          case 6
            call UI:Control_YesNO("确定需要关门吗？",l_bRes)
            if l_bRes
              call UI:Control_PanelMd("正在关闭门....")
              if x_b8Axis
                call IO:AxisDoor(false,true)
              else
                call IO:AxisDoor(false,false)
              endIf
            endIf
            cls()
          break

          //刷新当前轴值
          case 7


          break


        endSwitch


      break

      case -1

        if x_b8Axis
          call IO:Axis8Action(9)
        else
          call IO:Axis7Action(9)
        endIf

      break

    endSwitch



    //当前七轴位置
    if l_nKey!=-1 or !l_bFirst


      //


      l_bFirst=true
      gotoxy(0,0)
      put("运动机械手臂须上电     ")

      //××××××××××××××××××××××××××××


      sSItem[0]="位置mm   :"+toString(".3",l_nPosition)
      sSItem[1]="速度m/min:"+toString(".3",l_nSpeed)
      sSItem[2]="比例分度 :"+toString("",l_nPrecent)
      sSItem[3]="点动速度 :"+toString("",l_nJogSpeed)+"%"
      sSItem[4]="报警复位"
      sSItem[5]="门打开"
      sSItem[6]="门关闭"
      //sSItem[7]="当前马达值"
      if bCheckAxisSafte
        l_sBottom="+,-,,回零,运动,,,退出"
      else
        l_sBottom="+,-,记录,回零,运动,上传,保存,退出"
      endIf
      if !x_b8Axis

        call UI:Form_PanelList("LasMAN3.6->示教异步七轴","第七轴",sSItem,l_nIndex,l_sBottom)

      else
        call UI:Form_PanelList("LasMAN3.6->示教异步八轴","第八轴",sSItem,l_nIndex,l_sBottom)

      endIf


    endIf


    //报警处理
    if l_bAlarm
      call UI:Control_Mess("马达报警            ","")
    else
      if !l_bPowerOn
        if l_bBHome
          call UI:Control_Mess("马达已回零,未上电","")
        else
          call UI:Control_Mess("马达未回零,未上电","")
        endIf
      else
        if l_bBHome
          setTextMode(0)
          call UI:Control_Mess("马达已回零,已上电","")
        else
          call UI:Control_Mess("马达未回零,已上电","")
        endIf
      endIf

    endIf




    //2014.08.04
    //实时显示异步七轴八轴位置

    if l_bAlarm==false and l_bPowerOn==true
      if x_b8Axis
        call IO:GetAxis8Pos(l_nBuff,l_nPrecent)
      else
        call IO:GetAxis7Pos(l_nBuff,l_nPrecent)
      endIf
      gotoxy(0,2)
      put("轴当前位置:"+toString(".3",l_nBuff)+"     ")
    endIf
    delay(0)

  endWhile


end

--- TeachConfig.pgx ---
public program TeachConfig()
  local num l_nKey
  local num l_nPointIndex
  local bool l_bRes
  local string l_sBuff[2]
  local num l_nNum[40]
begin

  //配置示教


  //参数初始化



  title("LasMAN3.6->配置")
  call TxtFile:ReadCfg(l_bRes)
   IO:bWeldEnable=TxtFile:bWeldEnable
   IO:bExt7AxisEnable=TxtFile:b7Axis
   IO:bExt8AxisEnable=TxtFile:b8Axis
  if !l_bRes
    popUpMsg("读取配置文件不正确")
    return
  endIf
  l_sBuff[0]="关"
  l_sBuff[1]="开"
  //工具
  l_nNum[0]=TxtFile:tCfg.trsf.x
  l_nNum[1]=TxtFile:tCfg.trsf.y
  l_nNum[2]=TxtFile:tCfg.trsf.z
  l_nNum[3]=TxtFile:tCfg.trsf.rx
  l_nNum[4]=TxtFile:tCfg.trsf.ry
  l_nNum[5]=TxtFile:tCfg.trsf.rz

  //基本设置
  l_nNum[6]=TxtFile:nHomeSpeed
  l_nNum[7]=sel(TxtFile:bTeachToolMode,1,0)
  l_nNum[8]=sel(TxtFile:bMoveBack,1,0)

  //工艺
  l_nNum[9]=TxtFile:trPresetData.x
  l_nNum[10]=TxtFile:trPresetData.y
  l_nNum[11]=TxtFile:trPresetData.z
  l_nNum[12]=TxtFile:trPresetData.rx
  l_nNum[13]=TxtFile:trPresetData.ry



  //动作
  l_nNum[14]=TxtFile:trIODelay.x
  l_nNum[15]=TxtFile:trIODelay.y
  l_nNum[16]=TxtFile:trIODelay.rx
  //拐角
  l_nNum[17]=TxtFile:trCorner.z
  l_nNum[18]=TxtFile:trCorner.rx
  l_nNum[19]=TxtFile:trCorner.ry
  l_nNum[20]=TxtFile:trCorner.x


  l_nNum[21]=sel(TxtFile:b7Axis,1,0)
  l_nNum[22]=TxtFile:trAxisData.x
  l_nNum[23]=TxtFile:trAxisData.y
  l_nNum[24]=TxtFile:trAxisData.z



  l_nNum[25]=sel(TxtFile:bWeldEnable,1,0)
  l_nNum[26]=TxtFile:trIODelay.z
  // l_nNum[27]=sel(TxtFile:bStepMove,1,0)
  l_nNum[28]=TxtFile:nStepLength
  l_nNum[29]=DataBase:nRemoteProduct
  l_nNum[30]=sel(TxtFile:bMoreProd1Wp,1,0)
  l_nNum[27]=TxtFile:trIODelay.ry
  l_nNum[31]=sel(TxtFile:bAdjustSpEnable,1,0)

  //八轴
  l_nNum[32]=sel(TxtFile:b8Axis,1,0)
  l_nNum[33]=TxtFile:trAxisData.rx
  l_nNum[34]=TxtFile:trAxisData.ry
  l_nNum[35]=TxtFile:trAxisData.rz


   l_nNum[36]=sel(DataBase:bWpFinishIOOut,1,0)
   l_nNum[37]=sel(DataBase:bExtraContrAxis,1,0)
   l_nNum[38]=sel(DataBase:bThickPlate,1,0)


  cls()
  userPage()

  //******************
  //2013.11.14
  gotoxy(0,0)
  put("Val3版本号:")
  gotoxy(0,1)
  put(DataBase:sVersion[0])
  gotoxy(0,2)
  put("手臂类型:")
  gotoxy(0,3)
  put(DataBase:sVersion[1])
  gotoxy(0,4)
  put("安装方式:")
  gotoxy(0,5)
  put(DataBase:sVersion[2])
  gotoxy(0,6)
  put("控制器序号:")
  gotoxy(0,7)
  put(DataBase:sVersion[3])

  //********************
  call UI:Form_Config(l_nNum,l_nPointIndex)
  while true

    l_nKey=getKey()
    switch l_nKey


      //退出
      case 278
        call UI:Control_YesNO("确定要退出吗?",l_bRes)
        if l_bRes
          return
        endIf
      break


      //上传
      case 276
        call UI:Control_YesNO("确定要上传吗?",l_bRes)
        if l_bRes
          call Kit:UpLoad()
          //return
        endIf
      break

      case 277
        call UI:Control_YesNO("确定要保存吗?",l_bRes)
        if l_bRes
          TxtFile:tCfg.trsf.x  =    l_nNum[0]
          TxtFile:tCfg.trsf.y  =    l_nNum[1]
          TxtFile:tCfg.trsf.z  =    l_nNum[2]
          TxtFile:tCfg.trsf.rx  =    l_nNum[3]
          TxtFile:tCfg.trsf.ry  =    l_nNum[4]
          TxtFile:tCfg.trsf.rz  =    l_nNum[5]

          TxtFile:nHomeSpeed=l_nNum[6]
          TxtFile:bTeachToolMode=(l_nNum[7]==1)
          TxtFile:bMoveBack=(l_nNum[8]==1)

          //工艺
          //保证PWM频率低值为5，高值一定大于等于5
          TxtFile:trPresetData.y=max(5,l_nNum[10])
          TxtFile:trPresetData.x=max(TxtFile:trPresetData.y,l_nNum[9])

          TxtFile:trPresetData.z=max(0,l_nNum[11])
          TxtFile:trPresetData.rx=max(0,l_nNum[12])
          TxtFile:trPresetData.ry=max(0,l_nNum[13])



          //动作
          TxtFile:trIODelay.x=l_nNum[14]
          TxtFile:trIODelay.y=l_nNum[15]
          TxtFile:trIODelay.rx=l_nNum[16]
          //拐角
          TxtFile:trCorner.z=max(0,l_nNum[17])
          TxtFile:trCorner.rx=max(0,l_nNum[18])
          TxtFile:trCorner.ry=max(0,l_nNum[19])
          TxtFile:trCorner.x=round(min(max(0,l_nNum[20]),50))

          //7轴
          TxtFile:b7Axis=(l_nNum[21]==1)
          TxtFile:trAxisData.x=max(0,l_nNum[22])
          TxtFile:trAxisData.y=max(0,l_nNum[23])
          TxtFile:trAxisData.z=max(0,l_nNum[24])

          TxtFile:bWeldEnable=(l_nNum[25]==1)
          TxtFile:trIODelay.z=max(0,l_nNum[26])
          // TxtFile:bStepMove=(l_nNum[27]==1)
          TxtFile:nStepLength=max(0,l_nNum[28])
          DataBase:nRemoteProduct=l_nNum[29]
          TxtFile:bMoreProd1Wp=(l_nNum[30]==1)
          TxtFile:trIODelay.ry=max(0,l_nNum[27])
          TxtFile:bAdjustSpEnable=(l_nNum[31]==1)

          //8轴
          TxtFile:b8Axis=(l_nNum[32]==1)
          TxtFile:trAxisData.rx=max(0,l_nNum[33])
          TxtFile:trAxisData.ry=max(0,l_nNum[34])
          TxtFile:trAxisData.rz=max(0,l_nNum[35])


          //其他配置
          DataBase:bWpFinishIOOut=(l_nNum[36]==1)
          DataBase:bExtraContrAxis=(l_nNum[37]==1)
          DataBase:bThickPlate=(l_nNum[38]==1)








          call TxtFile:SaveCfg(l_bRes)
          if !l_bRes
            popUpMsg("保存出错")
          else
            popUpMsg("保存成功")
            //2014.2.17  在哪个坐标系中运动
            if !DataBase:bWorldMove
              $jogContext(TxtFile:tCfg,TxtFile:fArray,0)
            else
              $jogContext(TxtFile:tCfg,world,0)
            endIf
            DataBase:libSave()
          endIf
          cls()
          // return
        endIf
      break



      case 270
        switch l_nPointIndex
          case 7,8,21,25,30,31,32,36,37,38
            call UI:Sel_Edit(l_nNum[l_nPointIndex],32,min(10,l_nPointIndex+1),l_sBuff)
          break

          default
            call UI:Float_Edit(l_nNum[l_nPointIndex],32,min(10,l_nPointIndex+1))
          break
        endSwitch

      break



      case 261
        l_nPointIndex=l_nPointIndex-1
        if l_nPointIndex<0
          l_nPointIndex=38
        endIf

        // l_nPointIndex=max(0,l_nPointIndex-1)
      break


      case 266
        l_nPointIndex=l_nPointIndex+1
        if l_nPointIndex>38
          l_nPointIndex=0
        endIf
        // l_nPointIndex=min(35,l_nPointIndex+1)
      break

    endSwitch


    if  l_nKey!=-1
      call UI:Form_Config(l_nNum,l_nPointIndex)

    endIf


    delay(0)

  endWhile

end

--- TeachFrame.pgx ---
public program TeachFrame(frame& x_fFrame)
  local frame l_fFrame
  local point l_p[3]
  local num l_nIndex
  local num l_nKey
  local bool l_bRes
  local num l_nErr
  local frame l_fBuff
  local string l_sData[3]
  local trsf l_trFirst
begin

  //用户坐标系示教
  //link(l_fFrame,world)
  l_trFirst=x_fFrame.trsf
  l_fFrame=x_fFrame
  l_fBuff=x_fFrame
  l_fFrame.trsf={0,0,0,0,0,0}
  //2013.10.26
  // DataBase:fJogContext=x_fFrame
  link(DataBase:fJogContext,world)
  DataBase:fJogContext.trsf=position(l_fFrame,world)
  if DataBase:bWorldMove
    $jogContext(TxtFile:tCfg,world,0)
  else
    $jogContext(TxtFile:tCfg,DataBase:fJogContext,0)
  endIf
  //
  for l_nErr=0 to 2

    link(l_p[l_nErr],l_fFrame)
    l_p[l_nErr]=here(TxtFile:tCfg,l_fFrame)

  endFor

  resetMotion()

  resize(sSItem,1,6)
  l_sData[0]="原点"
  l_sData[1]="X方向点"
  l_sData[2]="Y方向点"

  sSItem[0]="X   :"+toString(".3",l_fBuff.trsf.x)
  sSItem[1]="Y   :"+toString(".3",l_fBuff.trsf.y)
  sSItem[2]="Z   :"+toString(".3",l_fBuff.trsf.z)
  sSItem[3]="RX  :"+toString(".3",l_fBuff.trsf.rx)
  sSItem[4]="RY  :"+toString(".3",l_fBuff.trsf.ry)
  sSItem[5]="RZ  :"+toString(".3",l_fBuff.trsf.rz)



  cls()
  userPage()
  if DataBase:nInterfaceType==5
    call UI:Form_LabelList("LasMAN3.6->坐标系示教","用户坐标系",sSItem,"参考点",l_sData,l_nIndex,"记录,对齐,测试,默认,,计算,保存,退出")
  else

    call UI:Form_LabelList("LasMAN3.6->坐标系示教","用户坐标系",sSItem,"参考点",l_sData,l_nIndex,"记录,对齐,测试,默认,上传,计算,保存,退出")

  endIf
  movej(l_p[0],TxtFile:tCfg,mNomSpeed)
  while  true
    l_nKey=getKey()
    switch l_nKey
      case 261
        // DataBase:fJogContext.trsf={0,0,0,0,0,0}
        // $jogContext(TxtFile:tCfg,DataBase:fJogContext,0)
        l_nIndex=max(l_nIndex-1,0)

        resetMotion()
        mNomSpeed.blend=off

        movej(l_p[l_nIndex],TxtFile:tCfg,mNomSpeed)

      break


      case 266
        //DataBase:fJogContext.trsf={0,0,0,0,0,0}
        //$jogContext(TxtFile:tCfg,DataBase:fJogContext,0)
        l_nIndex=min(l_nIndex+1,2)
        resetMotion()
        mNomSpeed.blend=off
        movej(l_p[l_nIndex],TxtFile:tCfg,mNomSpeed)


      break




      //记录
      case 271
        // $jogContext(TxtFile:tCfg,l_fFrame,0)
        call UI:Control_YesNO("确定要记录吗?",l_bRes)
        if l_bRes
          l_p[l_nIndex]=here(TxtFile:tCfg,l_fFrame)
        endIf
      break

      //对齐
      case 272
        //  $jogContext(TxtFile:tCfg,l_fFrame,0)
        call Kit:Align(TxtFile:tCfg)

      break

      //验证
      case 273
        // $jogContext(TxtFile:tCfg,l_fBuff,0)
        DataBase:fJogContext.trsf=  DataBase:fJogContext.trsf=position(l_fBuff,world)
        $jogContext(TxtFile:tCfg,DataBase:fJogContext,0)
      break

      case 274
        call UI:Control_YesNO("把默认值赋值给当前用户坐标系吗?",l_bRes)
        if l_bRes
          l_fBuff.trsf=TxtFile:trDefaultFrame
          sSItem[0]="X   :"+toString(".3",l_fBuff.trsf.x)
          sSItem[1]="Y   :"+toString(".3",l_fBuff.trsf.y)
          sSItem[2]="Z   :"+toString(".3",l_fBuff.trsf.z)
          sSItem[3]="RX  :"+toString(".3",l_fBuff.trsf.rx)
          sSItem[4]="RY  :"+toString(".3",l_fBuff.trsf.ry)
          sSItem[5]="RZ  :"+toString(".3",l_fBuff.trsf.rz)
        endIf
      break
      case 115
        call UI:Control_YesNO("把当前坐标系设为默认值吗?",l_bRes)
        if l_bRes
          TxtFile:trDefaultFrame=l_fBuff.trsf
        endIf
      break

      case 275
        if DataBase:nInterfaceType==10
          call UI:Control_YesNO("确定要上传吗?",l_bRes)
          if l_bRes
            call Kit:UpLoad()
          endIf


        endIf

      break


      //计算
      case 276
        call UI:Control_YesNO("确定要计算吗?",l_bRes)
        if l_bRes

          l_nErr=setFrame(l_p[0],l_p[1],l_p[2],l_fBuff)
          if l_nErr==-1
            popUpMsg("X方向点离原点太近")
          endIf
          if l_nErr==-2
            popUpMsg("Y方向点离原点太近")
          endIf
          sSItem[0]="X   :"+toString(".3",l_fBuff.trsf.x)
          sSItem[1]="Y   :"+toString(".3",l_fBuff.trsf.y)
          sSItem[2]="Z   :"+toString(".3",l_fBuff.trsf.z)
          sSItem[3]="RX  :"+toString(".3",l_fBuff.trsf.rx)
          sSItem[4]="RY  :"+toString(".3",l_fBuff.trsf.ry)
          sSItem[5]="RZ  :"+toString(".3",l_fBuff.trsf.rz)
        endIf
      break



      //保存
      case 277
        if l_trFirst==l_fBuff.trsf
          popUpMsg("没有计算")
        else
          call UI:Control_YesNO("确定要保存吗?",l_bRes)
          if l_bRes
            x_fFrame.trsf=l_fBuff.trsf
          endIf
        endIf
        cls()


      break




      //退出
      case 278
        call UI:Control_YesNO("确定要退出吗?",l_bRes)
        if l_bRes

          return
        endIf
      break

      //点位
      case 270
        call UI:Control_Point(l_p[l_nIndex])
      break

    endSwitch

    if l_nKey!=-1
      if DataBase:nInterfaceType==5
        call UI:Form_LabelList("LasMAN3.6->坐标系示教","用户坐标系",sSItem,"参考点",l_sData,l_nIndex,"记录,对齐,测试,默认,,计算,保存,退出")
      else

        call UI:Form_LabelList("LasMAN3.6->坐标系示教","用户坐标系",sSItem,"参考点",l_sData,l_nIndex,"记录,对齐,测试,默认,上传,计算,保存,退出")

      endIf
    endIf

    delay(0)

  endWhile







end

--- TeachHome.pgx ---
public program TeachHome()
  local num l_nKey
  local num l_nIndex
  local bool l_bRes
  local jointRx l_jJ
  local joint l_jJFirst
  local trsf l_trTrsf
begin
  //安全点示教

  //2014.07.28
  //同步七八轴
  if TxtFile:bSync7Axis or TxtFile:bSync8Axis
    if !ExtAxis:libExist("Disk://extAxisCan/extAxisCan.pjx")
      if ExtAxis:libLoad("Disk://extAxisCan/extAxisCan.pjx")!=0
        popUpMsg("加载外部轴出错")
        disablePower()
        return
      endIf
    endIf
  endIf



  resize(sSItem,1,6)
  l_jJ=TxtFile:jHome
  l_jJFirst=TxtFile:jHome
  sSItem[0]="J1:"+toString(".3",l_jJ.j1)
  sSItem[1]="J2:"+toString(".3",l_jJ.j2)
  sSItem[2]="J3:"+toString(".3",l_jJ.j3)
  sSItem[3]="J4:"+toString(".3",l_jJ.j4)
  sSItem[4]="J5:"+toString(".3",l_jJ.j5)
  sSItem[5]="J6:"+toString(".3",l_jJ.j6)

  cls()
  userPage()
  call UI:Form_PanelList("LasMAN3.6->示教安全点","安全点",sSItem,l_nIndex,"记录,,,,,上传,保存,退出")

  while DataBase:nInterfaceType==15
    l_nKey=getKey()
    switch l_nKey

      case 261
        l_nIndex=max(0,l_nIndex-1)
      break

      case 266
        l_nIndex=min(5,l_nIndex+1)
      break


      case  271

        call UI:Control_YesNO("确定要记录吗?",l_bRes)
        if l_bRes
          l_jJ=herej()
          sSItem[0]="J1:"+toString(".3",l_jJ.j1)
          sSItem[1]="J2:"+toString(".3",l_jJ.j2)
          sSItem[2]="J3:"+toString(".3",l_jJ.j3)
          sSItem[3]="J4:"+toString(".3",l_jJ.j4)
          sSItem[4]="J5:"+toString(".3",l_jJ.j5)
          sSItem[5]="J6:"+toString(".3",l_jJ.j6)
          //2014.12.04
          //记录七八轴的home位置
          if (TxtFile:bSync7Axis or TxtFile:bSync8Axis)
            call ExtAxis:RecordExtAxis(l_trTrsf,l_trTrsf,TxtFile:tCfg)
            TxtFile:trSync7Axis.y=l_trTrsf.x
            TxtFile:trSync8Axis.y=l_trTrsf.y
          endIf
        endIf
      break



      case 272

      break

      //上传
      case 276
        call UI:Control_YesNO("确定上传吗?",l_bRes)
        if l_bRes
          call Kit:UpLoad()
        endIf
      break


      //保存
      case 277
        if l_jJFirst==l_jJ
          popUpMsg("没有记录")
        else
          call UI:Control_YesNO("确定保存吗?",l_bRes)
          if l_bRes
            TxtFile:jHome=l_jJ

            call TxtFile:SaveCfg(l_bRes)
            if !l_bRes
              popUpMsg("保存失败")
            else
              popUpMsg("保存成功")
            endIf
          endIf
        endIf
      break


      //退出
      case 278
        call UI:Control_YesNO("确定退出吗?",l_bRes)
        if l_bRes
          return
        endIf
      break








    endSwitch
    if l_nKey!=-1 and l_nKey>260
      call UI:Form_PanelList("LasMAN3.6->示教安全点","安全点",sSItem,l_nIndex,"记录,,,,,上传,保存,退出")

    endIf

    //2014.7.30
    //同步七八轴
    if (TxtFile:bSync7Axis or TxtFile:bSync8Axis)
      call ExtAxis:RecordExtAxis(l_trTrsf,l_trTrsf,TxtFile:tCfg)
      gotoxy(0,12)
      put("七轴:"+toString(".3",l_trTrsf.x))
      if TxtFile:bSync8Axis
        gotoxy(20,12)
        put("八轴:"+toString(".3",l_trTrsf.y))
      endIf
    endIf

  endWhile

end

--- TeachNewTraj.pgx ---
public program TeachNewTraj()
  local bool l_bRes
  local num l_nType
  local num l_nNum
begin
  //示教路径
  //新建一条路径


  //初始化
  TxtFile:fTraj.trsf={0,0,0,0,0,0}
  TxtFile:fToffset.trsf={0,0,0,0,0,0}
  TxtFile:fArray.trsf={0,0,0,0,0,0}

  TxtFile:trWorkplace={0,0,0,0,0,1}
//  TxtFile:trDownLead=TxtFile:trDownleadData
//  TxtFile:trDownLead.ry=TxtFile:trDownLead.rz=0
  TxtFile:trArray={1,0,1,0,0,0}
  //参数初始化
  TxtFile:trPointCount={0,0,0,0,0,0}





  //圆的长度和圆弧度为0

  call UI:Form_SelSharp(TxtFile:nSingleType,l_bRes)
  if !l_bRes
    return
  endIf

//第一次示教点
bFirstTeach=false



 call TrajScreen()



end

--- TeachOffset.pgx ---
public program TeachOffset(frame& x_fOffset)
  local frame l_fFrame
  local point l_p[6]
  local num l_nIndex
  local num l_nKey
  local bool l_bRes
  local num l_nErr
  local frame l_fBuff[2]
  local string l_sData[6]
  local bool l_bOnePoint
  local trsf l_trTrsf
  local string l_sOorT
  local pointRx l_pP
  local num l_nDistance[2]
  local bool l_bFirst
  local point l_pF[2]
begin
  //l_trTrsf   临时偏差保存点
  //




  //安全机制
  resetMotion()
  userPage()
  cls()
  link(l_fFrame,world)
  //设置frame.进行验证

  //数据初始化
  link(l_fBuff[0],world)
  link(l_fBuff[1],world)

    link(l_pF[0],world)
  link(l_pF[1],world)


  l_fFrame=x_fOffset
  l_trTrsf=x_fOffset.trsf
  l_fFrame.trsf={0,0,0,0,0,0}


  //2013.10.28
  //DataBase:fJogContext=x_fOffset

  link(DataBase:fJogContext,world)
  DataBase:fJogContext.trsf=position(l_fFrame,world)

  if DataBase:bWorldMove
    $jogContext(TxtFile:tCfg,world,0)
  else
    $jogContext(TxtFile:tCfg,DataBase:fJogContext,0)
  endIf

  for l_nErr=0 to 5
    link(l_p[l_nErr],l_fFrame)
    l_p[l_nErr]=here(TxtFile:tCfg,l_fFrame)
  endFor


  //说明类型是三点法
  //给其赋值
  if TxtFile:nSingleType!=10 and TxtFile:nSingleType!=2 and TxtFile:nSingleType!=12 and size(TxtFile:pCut)>=3

    l_p[0]=TxtFile:pCut[0]
    l_p[1]=TxtFile:pCut[1]
    l_p[2]=TxtFile:pCut[2]
    l_bOnePoint=false
  endIf

  if DataBase:nInterfaceType==5 and  TxtFile:nSingleType==2 and TxtFile:nSingleType==12 and size(TxtFile:pCut)>=1

    l_p[0]=TxtFile:pCut[0]
    l_bOnePoint=true
  endIf

  if DataBase:nInterfaceType==11

    l_p[0].trsf=DataBase:trOffset[0]
    l_p[1].trsf=DataBase:trOffset[1]
    l_p[2].trsf=DataBase:trOffset[2]
    l_bOnePoint=false
  endIf



  //  //界面初始化
  //  l_sData[0]="X   :"+toString(".3",l_trTrsf.x)
  //  l_sData[1]="Y   :"+toString(".3",l_trTrsf.y)
  //  l_sData[2]="Z   :"+toString(".3",l_trTrsf.z)
  //  l_sData[3]="RX  :"+toString(".3",l_trTrsf.rx)
  //  l_sData[4]="RY  :"+toString(".3",l_trTrsf.ry)
  //  l_sData[5]="RZ  :"+toString(".3",l_trTrsf.rz)
  //
  //
  //  if l_bOnePoint
  //    resize(sSItem,1,2)
  //    sSItem[0]="标定点"
  //    sSItem[1]="修正点"
  //    // l_sData[2]="Y方向点"
  //    l_sOorT="一点法"
  //  else
  //    resize(sSItem,1,6)
  //    sSItem[0]="标定点1"
  //    sSItem[1]="标定点2"
  //    sSItem[2]="标定点3"
  //
  //    sSItem[3]="修正点1"
  //    sSItem[4]="修正点2"
  //    sSItem[5]="修正点3"
  //    l_sOorT="三点法"
  //  endIf
  //
  //  if DataBase:nInterfaceType==5
  //    call UI:Form_LabelList("LasMAN3.6->示教偏差","偏差值",l_sData,l_sOorT,sSItem,l_nIndex,"记录,计算,一点,三点,对齐,保存,数值,退出")
  //
  //  else
  //
  //    call UI:Form_LabelList("LasMAN3.6->示教偏差","偏差值",l_sData,l_sOorT,sSItem,l_nIndex,"记录,计算,一点,三点,对齐,保存,上传,退出")
  //
  //  endIf



  mNomSpeed.blend=off

  movej(l_p[l_nIndex],TxtFile:tCfg,mNomSpeed)
  //按键响应模式
  while  true
    l_nKey=getKey()
    switch l_nKey

      //向上
      case 261
        l_nIndex=max(l_nIndex-1,0)

        resetMotion()
        mNomSpeed.blend=off

        movej(l_p[l_nIndex],TxtFile:tCfg,mNomSpeed)

      break

      //向下
      case 266
        l_nIndex=min(l_nIndex+1,size(sSItem)-1)
        resetMotion()
        mNomSpeed.blend=off
        movej(l_p[l_nIndex],TxtFile:tCfg,mNomSpeed)


      break




      //记录
      case 271
        call UI:Control_YesNO("确定要记录吗?",l_bRes)
        if l_bRes
          l_p[l_nIndex]=here(TxtFile:tCfg,l_fFrame)
        endIf
      break



      //计算
      case 272
        l_nErr=0
        call UI:Control_YesNO("确定要计算吗?",l_bRes)
        if l_bRes
          if !l_bOnePoint
            if l_p[0].trsf==l_p[1].trsf or l_p[1].trsf==l_p[2].trsf or l_p[3].trsf==l_p[4].trsf or l_p[3].trsf==l_p[5].trsf
              popUpMsg("点没有完全记录")
              l_nErr=1
            else

              l_nErr=setFrame(l_p[0],l_p[1],l_p[2],l_fBuff[0])
              if l_nErr==-1
                popUpMsg("参考点X方向点离原点太近")
              endIf
              if l_nErr==-2
                popUpMsg("参考点Y方向点离原点太近")
              endIf

              if l_nErr==0
                l_nErr=setFrame(l_p[3],l_p[4],l_p[5],l_fBuff[1])
                if l_nErr==-1
                  popUpMsg("修正点X方向点离原点太近")
                else
                  if l_nErr==-2
                    popUpMsg("修正点Y方向点离原点太近")
                  else
                    //2014.3.7
                    //用来测试三点法
                    link(l_pF[0],l_fBuff[0])
                    link(l_pF[1],l_fBuff[1])
                    l_pF[0].trsf=l_pF[1].trsf={0,0,0,0,0,0}
                    l_trTrsf=position(l_pF[1],l_fFrame)*!(position(l_pF[0],l_fFrame))
                  endIf
                endIf
              endIf
            endIf

          else
            //作为偏差

            l_trTrsf=l_p[1].trsf*!l_p[0].trsf

          endIf

          //主要用来做提示用
          if l_nErr==0
            l_nDistance[0]=distance(world.trsf,l_trTrsf)
            if l_bOnePoint
              l_nDistance[1]=distance(l_p[0].trsf,l_p[1].trsf)
            else
              l_nDistance[1]=distance(l_p[0].trsf,l_p[3].trsf)
            endIf
            popUpMsg("原点间距离是"+toString(".3",l_nDistance[1])+",偏差距离是"+toString(".3",l_nDistance[0]))

          endIf
        endIf

      break

      //一点法
      case 273
        l_bOnePoint=true
        l_sOorT="一点法"

      break
      //三点法
      case 274
        l_bOnePoint=false
        l_sOorT="三点法"

      break
      //对齐
      case 275
        call Kit:Align(TxtFile:tCfg)

      break



      //保存
      case 276
        call UI:Control_YesNO("确定要保存吗?",l_bRes)
        if l_bRes
          x_fOffset.trsf=l_trTrsf
        endIf
      break


      case 277
        //示教局部时需要上传
        if DataBase:nInterfaceType==11
          call UI:Control_YesNO("确定要上传吗?",l_bRes)
          if l_bRes
            call Kit:UpLoad()
          endIf

        else
          l_pP.trsf=l_trTrsf
          call UI:Control_Point(l_pP)
          l_trTrsf=l_pP.trsf

        endIf
      break


      //退出
      case 278
        call UI:Control_YesNO("确定要退出吗?",l_bRes)
        if l_bRes

          return
        endIf
      break

      //点位
      case 270
        call UI:Control_Point(l_p[l_nIndex])
      break

    endSwitch



    //界面刷新
    if l_nKey!=-1 or !l_bFirst
      l_bFirst=true
      l_sData[0]="X   :"+toString(".3",l_trTrsf.x)
      l_sData[1]="Y   :"+toString(".3",l_trTrsf.y)
      l_sData[2]="Z   :"+toString(".3",l_trTrsf.z)
      l_sData[3]="RX  :"+toString(".3",l_trTrsf.rx)
      l_sData[4]="RY  :"+toString(".3",l_trTrsf.ry)
      l_sData[5]="RZ  :"+toString(".3",l_trTrsf.rz)
      if l_bOnePoint
        resize(sSItem,1,2)
        sSItem[0]="标定点"
        sSItem[1]="修正点"

      else
        resize(sSItem,1,6)
        sSItem[0]="标定点1"
        sSItem[1]="标定点2"
        sSItem[2]="标定点3"

        sSItem[3]="修正点1"
        sSItem[4]="修正点2"
        sSItem[5]="修正点3"
      endIf
      if DataBase:nInterfaceType==5
        call UI:Form_LabelList("LasMAN3.6->示教偏差","偏差值",l_sData,l_sOorT,sSItem,l_nIndex,"记录,计算,一点,三点,对齐,保存,数值,退出")

      else

        call UI:Form_LabelList("LasMAN3.6->示教偏差","偏差值",l_sData,l_sOorT,sSItem,l_nIndex,"记录,计算,一点,三点,对齐,保存,上传,退出")

      endIf




    endIf

    delay(0)

  endWhile

end

--- TeachPreset.pgx ---
public program TeachPreset()
  local num l_nKey
  local num l_nPointType
  local num l_nPointIndex
  local bool l_bRes
  local string l_sItemTitle
  local bool l_bKeyIO[3]
  local num l_nNum
  local bool l_bPower
  local bool l_bFirst
  local bool l_bLaserNoGas
  local bool l_bGunUp
begin
  //工艺示教
  //参数初始化
  DataBase:bStopPoll=true


  call TxtFile:ReadCfg(l_bRes)
   IO:bWeldEnable=TxtFile:bWeldEnable
   IO:bExt7AxisEnable=TxtFile:b7Axis
   IO:bExt8AxisEnable=TxtFile:b8Axis
  if !l_bRes
    popUpMsg("读取配置文件不正确")
    return
  endIf

  call TxtFile:ReadPreset(l_bRes)
  if !l_bRes
    popUpMsg("读取工艺文件不正确")
    return
  endIf

  if TxtFile:trPresetData.z<=0
    popUpMsg("配置中模拟量系数不能小于等于0")
    return
  endIf

  if TxtFile:trPresetData.x<=TxtFile:trPresetData.y
    popUpMsg("配置中PWM频率高不能小于等于PWM频率低")
    return
  endIf


  //轮询
  resize(sSItem,1,50)
  for l_nNum=0 to 49
    sSItem[l_nNum]="序号:"+toString("",l_nNum+1)
  endFor
  cls()
  DataBase:bStopPoll=false



  l_bGunUp=IO:bGunUp
  while true

    l_nKey=getKey()
    switch l_nKey

      //激光
      case 271


        if !isPowered() and !l_bKeyIO[0]
          popUpMsg("请先上电!")
        else
          l_bKeyIO[0]=!l_bKeyIO[0]
          if l_bKeyIO[0]
            if !l_bLaserNoGas
              l_bKeyIO[2]=true
            endIf
          endIf
          call IO:KeyDigtalIO(l_bKeyIO[2],l_bKeyIO[1],l_bKeyIO[0],0,0)
        endIf

      break






      //随动
      case 272
        IO:bGunUp=false
        if !isPowered() and !l_bKeyIO[1]
          popUpMsg("请先上电!")
        else
          l_bKeyIO[1]=!l_bKeyIO[1]
          call IO:KeyDigtalIO(l_bKeyIO[2],l_bKeyIO[1],l_bKeyIO[0],0,0)
        endIf
      break

      //气体
      case 273

        if !isPowered() and !l_bKeyIO[2]
          popUpMsg("请先上电!")
        else
          if !l_bKeyIO[0]
            l_bKeyIO[2]=!l_bKeyIO[2]
          endIf
          call IO:KeyDigtalIO(l_bKeyIO[2],l_bKeyIO[1],l_bKeyIO[0],0,0)
        endIf
      break


      //上传
      case 275
        call UI:Control_YesNO("确定要上传吗?",l_bRes)
        if l_bRes
          call Kit:UpLoad()
        endIf
      break


      //退出
      case 278
        IO:bGunUp=l_bGunUp
        call UI:Control_YesNO("确定要退出吗?",l_bRes)
        if l_bRes
          return
        endIf
      break


      //修改
      case 276,270
        call UI:Control_Preset(TxtFile:nPreset,l_nPointIndex+1)
        cls()
      break




      case 277
        call UI:Control_YesNO("确定要保存吗?",l_bRes)
        if l_bRes
          call TxtFile:SavePreset(l_bRes)
          if !l_bRes
            popUpMsg("保存出错")
          else
            popUpMsg("保存成功")
          endIf
          cls()
        endIf
      break



      case 261
        l_nPointIndex=max(0,l_nPointIndex-1)
      break


      case 266
        l_nPointIndex=min(size(sSItem)-1,l_nPointIndex+1)
      break

      //q
      //开光时不强制开气
      case 113
        call UI:Control_YesNO("确定需要开光时不强制开气",l_bRes)
        l_bLaserNoGas=l_bRes

      break


      //97
      case 97
        call UI:Control_YesNO("确定需要开随动不抬枪",l_bRes)
        IO:bGunUp=!l_bRes
      break

    endSwitch


    if (l_nKey<279  and l_nKey>=260) or isPowered()!=l_bPower or !l_bFirst or l_nKey==113 or l_nKey==97
      l_bPower=isPowered()
      if !l_bPower
        l_bKeyIO[0]=l_bKeyIO[1]=l_bKeyIO[2]=false
      endIf
      l_bFirst=true




      //IO配置
      call IO:Preset(TxtFile:nPreset,l_nPointIndex+1,TxtFile:trPresetData.z,TxtFile:trPresetData.x,TxtFile:trPresetData.y)
      call IO:GetPreset(DataBase:nPresetData,TxtFile:trPresetData.z,TxtFile:trPresetData.x,TxtFile:trPresetData.y)
      call UI:Form_Simulation("LasMAN3.6->示教工艺","工艺表",sSItem,l_nPointIndex,DataBase:nPresetData,l_bKeyIO)


      gotoxy(0,0)
      put("测试请上电!")

      //2014.06.06
      if l_bGunUp
        gotoxy(0,1)
        put("q->开光不开气")
        gotoxy(0,2)
        put("a->随动不抬枪")

      endIf
      if l_bLaserNoGas
        gotoxy(0,3)
        put("激光与气体不联动")
      endIf



    endIf




    delay(0)


  endWhile

end

--- TeachProduct.pgx ---
public program TeachProduct()
  local num l_nKey
  local bool l_bRes
  local string l_sProductName
  local bool l_bPause
  local string l_sBottom
  local jointRx l_jJ
  local bool l_bPauseStauts
  local string l_sA
  local num l_nWeld
  local bool l_bWeld
begin
  //生产模式
  //是否在零位

  //初始化
  cls()
  resetMotion()
  resize(sSItem,1,12)
  resize(sMess,1,11)

  //检查条件
  DataBase:nToolMode=workingMode()
  if DataBase:nToolMode!=4
    popUpMsg("机器手臂请切换到远程模式")
    return
  endIf


  call UI:Control_PanelMd("请等待,正在载入库......")
  DataBase:bStopPoll=true

  //检查机械手臂是否在零位
  l_jJ=herej()
  l_nKey= abs(l_jJ.j1-TxtFile:jHome.j1)+abs(l_jJ.j2-TxtFile:jHome.j2)+abs(l_jJ.j3-TxtFile:jHome.j3)
  l_nKey=l_nKey+ abs(l_jJ.j4-TxtFile:jHome.j4)+abs(l_jJ.j5-TxtFile:jHome.j5)+abs(l_jJ.j6-TxtFile:jHome.j6)
  if l_nKey>0.3
    popUpMsg("请回到零位")
    return
  endIf





  //可以生产的部分为空
  //  for l_nKey=0 to 9
  //    DataBase:bCanProduct[l_nKey]=false
  //  endFor

  //检查文件是否正确
  call TxtFile:IsFileOK(l_bRes)
  if !l_bRes
    //popUpMsg("读取辅助文件出错")
    return
  endIf

  //如果只有一个工位，则文件预读
  if DataBase:nWorkPlaceCount==1 and !TxtFile:bMoreProd1Wp
    call GetProductMess("只有一个工位，预读取文件")
    call TxtFile:ReadProduct("Disk://Txt/Product1.txt",DataBase:sProductName[1],false,l_bRes)
    if !l_bRes
      popUpMsg("读取生产文件出错")
      return
    endIf


    if TxtFile:bMatchPreset
      call TxtFile:ReadMatchPreset("Disk://Txt/Preset1.txt",TxtFile:sPresetName[0],l_bRes)
      if !l_bRes
        popUpMsg("读取工艺文件出错")
        return
      endIf
    endIf
  endIf



  //界面初始化

  bPowerFlag=false
  //初始化消息
  for l_nKey=0 to 10
    sSItem[l_nKey]=""
    sMess[l_nKey]=""
  endFor

  if TxtFile:bWeldEnable
    l_sA="回退"
  else
    l_sA=""
  endIf

  //生产模式记录
  if TxtFile:bMoreProd1Wp
    logMsg("生产模式:同工位多产品")
  else
    switch DataBase:nCycleMode
      case 0
        logMsg("生产模式:按钮触发单工位")
      break

      case 1
        logMsg("生产模式:按钮触发单周期")
      break

      case 2
        logMsg("生产模式:按钮触发多周期")
      break
      case 3
        logMsg("生产模式:无需按钮触发")
      break

      case 4
        logMsg("生产模式:排队")
      break
      case 5
        logMsg("生产模式:自定义")
      break
    endSwitch
  endIf


  DataBase:bStopPoll=false
  taskCreate "Product",100,Product()

  cls()
  wait(getKey()==-1)
  while  DataBase:nInterfaceType==13
    call GetListItems()

    //机械手臂掉电了
    DataBase:bPowerOn=isPowered()
    bPowerFlag=DataBase:bPowerOn or bPowerFlag
    if DataBase:bPowerOn==false and bPowerFlag
      logMsg("机械手臂掉电")
      taskSuspend("Product")
      stopMove()
      call IO:SafteyIO()
      l_bPause=true
      bPowerFlag=false
      call GetProductMess("机械手臂掉电")
    endIf

    //IO轮询
    call IO:ProductPoll(DataBase:nCycleCount,DataBase:nInterfaceType,l_bPause)

    //停止信号被触发
    if  DataBase:nInterfaceType!=13
      call UI:Control_PanelMd("停止信号被触发......")
      delay(2)
    endIf

    //暂停信号
    if l_bPause!=l_bPauseStauts
      l_bPauseStauts=l_bPause
      if l_bPause
        stopMove()
        if taskStatus("Product")==1
          taskSuspend("Product")
        endIf
        stopMove()
        call IO:SafteyIO()
        call IO:Light(0)

      else

        //2014.02.03
        //为同步外部轴设置
        if DataBase:nPointType==2 and TxtFile:trWorkplace.rz!=-1
          if !TxtFile:bWeldEnable or (TxtFile:bWeldEnable and !DataBase:bIOControl)

            call IO:Preset(TxtFile:nPreset,TxtFile:trWorkplace.rz,TxtFile:trPresetData.z,TxtFile:trPresetData.x,TxtFile:trPresetData.y)
            call IO:PerforatiAction(TxtFile:trIODelay.x,TxtFile:trIODelay.y)
          endIf
        endIf
        if taskStatus("Product")==0
          taskResume("Product",0)

        endIf
        restartMove()
        call IO:Light(2)
      endIf
    endIf


    //查询按钮
    l_nKey=getKey()
    switch l_nKey


      //暂停与继续
      case 271
        if !l_bPause
          l_bPause=!l_bPause
        else
          if !isPowered()
            popUpMsg("请先上电")
          else
            call UI:Control_YesNO("确定要继续吗?",l_bRes)
            if l_bRes
              call GetProductMess("机械手臂继续")
              l_bPause=!l_bPause
            endIf
          endIf
        endIf
      break

      //上电
      case 272
        if isPowered()
          bPowerFlag=true
        else
          call UI:Control_YesNO("确定要上电吗?",l_bRes)
          call UI:Form_Product("LasMAN3.6->生产界面",sMess,sSItem,l_sBottom)
          if l_bRes
            if DataBase:nToolMode!=4
              popUpMsg("机器手臂请切换到远程模式")
            else
              enablePower()

              if !watch(isPowered(),5)
                popUpMsg("上电失败，检查急停按钮")
              else
                logMsg("上电")
                bPowerFlag=true
                call GetProductMess("机械手臂上电")
              endIf
            endIf
          endIf
        endIf
      break



      //在焊接下进行回退
      case 273
        if TxtFile:bWeldEnable
          if !l_bPause or TxtFile:trPointCount.y>500
            popUpMsg("机械手臂只能在暂停状态下与焊接点小于500回退")

          else
            if DataBase:nPointType!=2
              popUpMsg("机械手臂不在焊接状态")
            else
              if !l_bWeld
                call UI:Control_YesNO("确定需要回退吗",l_bRes)
                if l_bRes
                  call GetProductMess("执行回退程序")
                  disablePower()
                  call GetProductMess("计算回退路径")
                  logMsg("执行回退")
                  call WeldTraj(l_bRes)
                  if !l_bRes
                    popUpMsg("回退路径计算失败")
                  else
                    if taskStatus("Product")!=-1
                      taskKill("Product")
                      wait(taskStatus("Product")==-1)
                    endIf
                    call GetProductMess("程序开始执行")
                    taskCreate "Product",100,Motion:TeachSimu(0,0)
                    l_bWeld=true
                  endIf
                endIf
              else
                popUpMsg("已执行回退算法")
              endIf

            endIf
          endIf
        endIf
      break


      //退出
      case 278
        call UI:Control_YesNO("确定要退出吗?",l_bRes)
        if l_bRes
          logMsg("退出生产程序")
          DataBase:nInterfaceType=9
        endIf
      break


    endSwitch


    //界面

    if !l_bPause
      l_sBottom="暂停,上电,"+l_sA+",,,,,退出"
    else
      l_sBottom="继续,上电,"+l_sA+",,,,,退出"
    endIf
    call UI:Form_Product("LasMAN3.6->生产界面",sMess,sSItem,l_sBottom)
    gotoxy(32,0)


    //暂停与继续状态确认
    if !l_bPause
      l_bWeld=false
      setTextMode(0)
      put("     ")
      //只有排队模式才会去检查按钮信号
      if DataBase:nCycleMode==4
        call IO:CanProduct(DataBase:nWorkPlaceButto)
      endIf
    else
      setTextMode(3)
      put("已暂停")
    endIf




    delay(0)

  endWhile




  //生产结束
  DataBase:bMoveTask=false
  if taskStatus("ReadFile")!=-1
    taskKill("ReadFile")
  endIf

  if taskStatus("Preset")!=-1
    taskKill("Preset")
  endIf
  if taskStatus("Product")!=-1
    taskKill("Product")
  endIf
  if taskStatus("WeldEnd")!=-1
    taskKill("WeldEnd")
  endIf
  call Motion:KillTask()
  call UI:Control_PanelMd("生产结束......")
  DataBase:nWorkPlaceButto=-1
  delay(2)

end

--- TeachRecipe.pgx ---
public program TeachRecipe()
  local num l_nKey
  local bool l_bRes
  local bool l_bFirst
  local num l_nMonitor
begin

  //下位机对于产品编辑主界面
  //包括删除，示教，模拟，调图

  resetMotion()

  DataBase:bStopPoll=true
  call TxtFile:ReadCfg(l_bRes)
  IO:bWeldEnable=TxtFile:bWeldEnable
  IO:bExt7AxisEnable=TxtFile:b7Axis
  IO:bExt8AxisEnable=TxtFile:b8Axis
  if !l_bRes
    popUpMsg("读取配置文件出错")
    return
  endIf
  call TxtFile:ReadProductName("Disk://Txt/Recipe.txt",l_bRes)
  if !l_bRes
    popUpMsg("读取产品名出错")
    return
  endIf
  call TxtFile:ReadProduct("Disk://Txt/Recipe.txt",TxtFile:sProductName,true,l_bRes)
  DataBase:sProductName=TxtFile:sProductName
  if !l_bRes
    if TxtFile:tCfg.trsf!=TxtFile:tFileTool.trsf
      popUpMsg("产品的工具不一致")
    else
      popUpMsg("读取生产文件出错")
    endIf
    return
  endIf

  call TxtFile:ReadAction(l_bRes)
  if !l_bRes
    popUpMsg("读取动作文件出错")
    return
  endIf
  call TxtFile:ReadPreset(l_bRes)
  if !l_bRes
    popUpMsg("读取工艺文件出错")
    return
  endIf
  cls()

  //2014.07.28
  //同步七八轴
  if TxtFile:bSync7Axis or TxtFile:bSync8Axis
    if !ExtAxis:libExist("Disk://extAxisCan/extAxisCan.pjx")
      if ExtAxis:libLoad("Disk://extAxisCan/extAxisCan.pjx")!=0
        popUpMsg("加载外部轴出错")
        disablePower()
        return
      endIf
    endIf
  endIf


  DataBase:bStopPoll=false

  //第七或者8轴到达安全点

  if TxtFile:b7Axis and ((DataBase:nWorkPlaceIndex==1 and DataBase:bMutexAxis) or !DataBase:bMutexAxis)
    bCheckAxisSafte=true
    call TeachAxis(TxtFile:trAxisData.x,TxtFile:trAxisData.y,TxtFile:trAxisData.z,TxtFile:trAxisData.rx,false)
    bCheckAxisSafte=false
    call IO:Axis7onPosition(TxtFile:trAxisData.x,TxtFile:trAxisData.z,l_bRes)
    if !l_bRes
      popUpMsg("异步外部7轴没有处在安全点")
      return
    endIf
  endIf

  if TxtFile:b8Axis  and ((DataBase:nWorkPlaceIndex==2 and DataBase:bMutexAxis) or !DataBase:bMutexAxis)
    bCheckAxisSafte=true
    call TeachAxis(TxtFile:trAxis8Data.x,TxtFile:trAxis8Data.y,TxtFile:trAxis8Data.z,TxtFile:trAxis8Data.rx,true)
    bCheckAxisSafte=false
    call IO:Axis8onPosition(TxtFile:trAxis8Data.x,TxtFile:trAxis8Data.z,l_bRes)
    if !l_bRes
      popUpMsg("异步外部8轴没有处在安全点")
      return
    endIf
  endIf








  while  DataBase:nInterfaceType==5
    for l_nKey=0 to size(TxtFile:nPartTrajCount)-1
      TxtFile:nPartTrajCount[l_nKey]=0
    endFor
    bSaveTxt=false
    l_nKey=getKey()

    switch l_nKey
      case 261
        if TxtFile:nTotalTraj>1
          nTrajIndex=nTrajIndex-1
        endIf
      break


      case 266
        if TxtFile:nTotalTraj>1
          nTrajIndex=nTrajIndex+1
        endIf
      break


      //回零
      case 271

        call Kit:GoHome()
      break

      //示教
      case 272
        //2015.09.08
        //对序号进行初始化
        nApproIndex=nLeaveIndex=nCutIndex=0
        TxtFile:nTrajIndex=TxtFile:nTotalTraj+1
        call TeachNewTraj()
        nTrajIndex=TxtFile:nTotalTraj-1
        cls()
      break

      //模拟
      case 273
        if TxtFile:nTotalTraj<1
          popUpMsg("产品没有路径")
        else
          call UI:Control_YesNO("确定要模拟吗?",l_bRes)
          if l_bRes
            DataBase:bKeyIO[0]= DataBase:bKeyIO[1]= DataBase:bKeyIO[2]=false
            TxtFile:nTrajIndex=nTrajIndex+1
            call Simulate(nTrajIndex+1)
            call UI:Control_PanelMd("模拟结束")
            DataBase:bKeyIO[0]= DataBase:bKeyIO[1]= DataBase:bKeyIO[2]=false
            delay(1)
            cls()

          endIf
        endIf
      break


      //开始整体模拟


      case 113
        if TxtFile:nTotalTraj<1
          popUpMsg("产品没有路径")
        else
          call UI:Control_YesNO("确定要从当前路径模拟吗?",l_bRes)
          if l_bRes
            DataBase:bKeyIO[2]=DataBase:bKeyIO[1]=DataBase:bKeyIO[0]=false
            DataBase:bStopSimul=false
            while nTrajIndex<TxtFile:nTotalTraj and DataBase:bStopSimul==false
              TxtFile:nTrajIndex=nTrajIndex+1
              call Simulate(nTrajIndex+1)

              nTrajIndex=nTrajIndex+1
            endWhile
            DataBase:bKeyIO[2]=DataBase:bKeyIO[1]=DataBase:bKeyIO[0]=false
            call UI:Control_PanelMd("模拟结束")
            delay(1)
            cls()
          endIf
        endIf

      break




      //对齐
      case 276
        call UI:Control_YesNO("确定要对齐吗?",l_bRes)
        if l_bRes
          call Kit:Align(TxtFile:tCfg)
          cls()
        endIf

      break



      //调图
      case 274,270
        if TxtFile:nTotalTraj<1
          popUpMsg("产品没有路径")
        else
          //2015.12.30
          //安全因素进行切换
          while workingMode()!=1
            popUpMsg("请先切换到手动模式,然后点击OK")
            delay(0.1)
          endWhile


          call UI:Control_YesNO("确定要调图吗?",l_bRes)
          if l_bRes
            //2015.09.08
            //对序号进行初始化
            nApproIndex=nLeaveIndex=nCutIndex=0
            TxtFile:nTrajIndex=nTrajIndex+1
            call AdjustTraj(nTrajIndex+1)
            cls()
          endIf
        endIf
      break

      //删除
      case 275
        DataBase:bStopPoll=true
        if TxtFile:nTotalTraj<1
          popUpMsg("产品没有路径")
        else
          call UI:Control_YesNO("确定要删除路径吗?",l_bRes)
          if l_bRes
            call UI:Control_PanelMd("请等待,正在删除......")
            call TxtFile:EditRecipe(nTrajIndex+1,true,l_bRes)
            if !l_bRes
              popUpMsg("删除文件出错")
            else
              call TxtFile:ReadProduct("Disk://Txt/Recipe.txt",TxtFile:sProductName,true,l_bRes)
              if !l_bRes
                popUpMsg("读取生产文件出错")
                return
              endIf
            endIf
          endIf
        endIf
        cls()
      break




      //上传
      case 277
        if TxtFile:nTotalTraj<1
          popUpMsg("产品没有路径")
        else
          call UI:Control_YesNO("确定要上传吗?",l_bRes)
          if l_bRes

            call Kit:UpLoad()
            //return
          endIf
        endIf
      break

      //退出
      case 278,255
        call UI:Control_YesNO("确定要退出吗?",l_bRes)
        if l_bRes
          return
        endIf
      break



      //112
      //修改产品的坐标系与偏差
      case 112
        call UI:Control_Recipe(TxtFile:fProduct.trsf,TxtFile:fPofffset.trsf)
      break




    endSwitch

    if l_nKey!=-1  or !l_bFirst
      l_bFirst=true

      //2015.5.21
      TxtFile:trPointCount={0,0,0,0,0,0}
      resetMotion()
      //  call UI:Form_PanelList("LasMAN3.6->编辑产品","路径列表",TxtFile:sTrajName,nTrajIndex,"回零,新建,模拟,调图,删除,对齐,上传,退出")
      call UI:Form_PanelList("LasMAN3.6->编辑产品","路径列表",TxtFile:sTrajNameType,nTrajIndex,"回零,新建,模拟,调图,删除,对齐,上传,退出")
      call UI:Control_LeftCut(0)


      if TxtFile:nTotalTraj>=1
        nTrajIndex=max(0,nTrajIndex)
        TxtFile:nSingleType=TxtFile:nTrajType[nTrajIndex]
        call UI:Control_Mess("产品名称:"+TxtFile:sProductName,toString("",nTrajIndex+1)+"->"+left(TxtFile:sTrajType[TxtFile:nSingleType]+"            ",12))
      else
        call UI:Control_Mess("产品名称:"+TxtFile:sProductName,"")

      endIf
    endIf
    DataBase:bStopPoll=false
    delay(0)

  endWhile



end

--- TeachRemote.pgx ---
public program TeachRemote()
  local num l_nIndex
  local num l_nKey
  local bool l_bRes
  local bool l_bUFile
  local string l_sSFileName
  local joint l_jJ
  local bool l_bFirst
begin
  //远程模式
  //不需要上位机来进行产品的生产


  //安全机制
  resetMotion()




  //是否在零位
  l_jJ=herej()
  l_nKey= abs(l_jJ.j1-TxtFile:jHome.j1)+abs(l_jJ.j2-TxtFile:jHome.j2)+abs(l_jJ.j3-TxtFile:jHome.j3)
  l_nKey=l_nKey+abs(l_jJ.j4-TxtFile:jHome.j4)+abs(l_jJ.j5-TxtFile:jHome.j5)+abs(l_jJ.j6-TxtFile:jHome.j6)
  if l_nKey>0.1
    popUpMsg("请回到零位")
    return
  endIf


  if DataBase:nToolMode!=4
    popUpMsg("请切换到远程模式")
    return
  endIf

  //同工位多产品不支持远程生产
  if TxtFile:bMoreProd1Wp
    popUpMsg("同工位多产品模式不支持远程生产")
    return
  endIf

  //界面初始化

  resize(sMess,1,1)
  sMess[0]=""
  DataBase:nCycleCount=1
  DataBase:nWorkPlaceCount=0
  DataBase:bStopPoll=true
  if $fileExists("Disk://Txt/Recipe.txt")
    $copy("Disk://Txt/Recipe.txt","Disk://OffTxt/Recipe.txt")
  endIf

  if $fileExists("Disk://Txt/Product1.txt")
    $copy("Disk://Txt/Product1.txt","Disk://OffTxt/Product1.txt")
  endIf

  if $fileExists("Disk://Txt/Product2.txt")
    $copy("Disk://Txt/Product2.txt","Disk://OffTxt/Product2.txt")
  endIf
  if $fileExists("Disk://Txt/Product3.txt")
    $copy("Disk://Txt/Product3.txt","Disk://OffTxt/Product3.txt")
  endIf

  if $fileExists("Disk://Txt/Product4.txt")
    $copy("Disk://Txt/Product4.txt","Disk://OffTxt/Product4.txt")
  endIf
  if !libList("Disk://OffTxt",sSItem)
    popUpMsg("路径不存在")
    return
  endIf
  cls()

  DataBase:bStopPoll=false

  //按键响应模式
  while  true
    l_nKey=getKey()
    switch l_nKey

      //向上
      case 261
        l_nIndex=max(l_nIndex-1,0)


      break

      //向下
      case 266
        l_nIndex=min(l_nIndex+1,size(sSItem)-1)


      break




      //添加
      case 271
        DataBase:bStopPoll=true
        if size(sMess)>=4
          popUpMsg("工位数不能超过4个")
        else
          if (size(sSItem)==1 and sSItem[0]=="") or l_nIndex==-1
            popUpMsg("没有文件")
          else
            call UI:Control_YesNO("确定要添加吗?",l_bRes)

            if l_bRes
              call UI:Control_PanelMd("请等待,正在配置文件......")
              if l_bUFile

                l_sSFileName="USB0://"+sSItem[l_nIndex]

              else

                l_sSFileName="Disk://OffTxt/"+sSItem[l_nIndex]
              endIf

              //查看一般情况是否有问题
              call TxtFile:ReadProductName(l_sSFileName,l_bRes)
              if !l_bRes
                popUpMsg("文件不符合规范")
              else
                //查看tool是否是一样
                call TxtFile:ReadProduct(l_sSFileName,TxtFile:sProductName,false,l_bRes)
                if !l_bRes  or  TxtFile:nTotalTraj<1
                  popUpMsg("文件不符合规范")
                else
                  if sMess[0]==""
                    DataBase:nWorkPlaceCount=1
                  else
                    DataBase:nWorkPlaceCount=size(sMess)+1
                  endIf

                  resize(sMess,1,DataBase:nWorkPlaceCount)
                  sMess[DataBase:nWorkPlaceCount-1]="工位"+toString("",DataBase:nWorkPlaceCount)+":"+TxtFile:sProductName
                  DataBase:sProductName[DataBase:nWorkPlaceCount]=TxtFile:sProductName
                  call TxtFile:BackupProduct(l_sSFileName,DataBase:nWorkPlaceCount,false)
                endIf
              endIf
            endIf
          endIf
        endIf
        cls()
      break



      //删除
      case 272
        if DataBase:nWorkPlaceCount==0
          popUpMsg("工位已清空")
        else
          call UI:Control_YesNO("确定要删除吗?",l_bRes)
          if l_bRes
            if DataBase:nWorkPlaceCount==1
              resize(sMess,1,1)
              sMess[0]=""
            else
              resize(sMess,1,DataBase:nWorkPlaceCount-1)

            endIf
            DataBase:nWorkPlaceCount=DataBase:nWorkPlaceCount-1
          endIf
        endIf
      break


      //U盘
      case 273
        l_bUFile=true
        if !libList("USB0://",sSItem)
          popUpMsg("路径不存在")
        endIf


      break
      //CS8C
      case 274
        l_bUFile=false
        if !libList("Disk://OffTxt",sSItem)
          popUpMsg("路径不存在")
          return
        endIf

      break
      //参数
      case 275
        //  call UI:control
        call UI:Control_Remote(DataBase:nCycleMode,DataBase:nCycleCount)
      break



      //生产
      case 277
        call UI:Control_YesNO("确定要生产吗?",l_bRes)
        if l_bRes
          disablePower()
          if DataBase:nWorkPlaceCount<1 or DataBase:nWorkPlaceCount>4
            popUpMsg("工位个数不正确!")
          else
            cls()
            call UI:Control_PanelMd("请等待,正在载入库......")
            for l_nIndex=1 to DataBase:nWorkPlaceCount
              call TxtFile:BackupProduct("",l_nIndex,true)

            endFor
            DataBase:nInterfaceType=13
            call TeachProduct()
            return

          endIf

        endIf
      break




      //退出
      case 278
        call UI:Control_YesNO("确定要退出吗?",l_bRes)
        if l_bRes

          return
        endIf
      break

    endSwitch



    //界面刷新
    if (l_nKey>0 and l_nKey<279) or !l_bFirst
      l_bFirst=true
      if l_bUFile
        call UI:Form_LabelList("LasMAN3.6->远程生产","工位信息",sMess,"U盘文件",sSItem,l_nIndex,"添加,删除,U盘,CS8C,配置,,生产,退出")

      else
        call UI:Form_LabelList("LasMAN3.6->远程生产","工位信息",sMess,"控制器文件",sSItem,l_nIndex,"添加,删除,U盘,CS8C,配置,,生产,退出")

      endIf



    endIf

    delay(0)
    DataBase:bStopPoll=false
  endWhile







end

--- TeachSyncAxis.pgx ---
public program TeachSyncAxis()
  local num l_nKey
  local bool l_bRes
  local num l_nIndex
  local bool l_bFirst
  local num l_nBuff
  local string l_sBottom
  local trsf l_trExtAxis
  local string l_sS[2]
  local point l_p
begin

  //示教同步七八轴
  resetMotion()
  call TxtFile:ReadCfg(l_bRes)
  IO:bWeldEnable=TxtFile:bWeldEnable
  IO:bExt7AxisEnable=TxtFile:b7Axis
  IO:bExt8AxisEnable=TxtFile:b8Axis
  if !l_bRes
    popUpMsg("读取配置文件不正确")
    return
  endIf
  wait(isKeyPressed(272)==false)

  //2014.07.28
  //同步七八轴
  if TxtFile:bSync7Axis or TxtFile:bSync8Axis
    if !ExtAxis:libExist("Disk://extAxisCan/extAxisCan.pjx")
      if ExtAxis:libLoad("Disk://extAxisCan/extAxisCan.pjx")!=0
        popUpMsg("加载外部轴出错")
        return
      endIf
    endIf
  endIf


  cls()

  resize(sSItem,1,2)
  l_sS[1]="开"
  l_sS[0]="关"
  l_trExtAxis.x=TxtFile:trSync7Axis.y
  l_trExtAxis.y=TxtFile:trSync8Axis.y


  //l_trExtAxis.rx=TxtFile:trSync7Axis.x
  // l_trExtAxis.ry=TxtFile:trSync8Axis.x

  while  DataBase:nInterfaceType==19 or DataBase:nInterfaceType==18


    //判断按键是否一直按着
    l_nKey=getKey()



    switch l_nKey


      case 261
        l_nIndex=max(0,l_nIndex-1)

      break

      //向下
      case 266
        l_nIndex=min(6,l_nIndex+1)
      break


      //参考
      case 271
        if TxtFile:bSync7Axis==false and TxtFile:bSync8Axis==false
          popUpMsg("同步七八轴未配置")
        else
          call UI:Control_YesNO("确定需要设置参考位吗？",l_bRes)
          if l_bRes
            //call ExtAxis:Reset()
            call ExtAxis:homing(ExtAxis:nAxesSum,l_bRes)
            if l_bRes
              popUpMsg("设置成功")
            else
              popUpMsg("设置失败")
            endIf
          endIf
        endIf

      break



      //复位
      case 272
        if TxtFile:bSync7Axis==false and TxtFile:bSync8Axis==false
          popUpMsg("同步七八轴未配置")
        else
          call UI:Control_YesNO("确定需要复位吗？",l_bRes)
          if l_bRes
            call ExtAxis:Reset()
          endIf
        endIf

      break




      //记录
      case 273

        if TxtFile:bSync7Axis==false and TxtFile:bSync8Axis==false
          popUpMsg("同步七八轴未配置")
        else
          call UI:Control_YesNO("确定需要记录吗？",l_bRes)
          if l_bRes
            call ExtAxis:RecordExtAxis(l_trExtAxis,l_trExtAxis,TxtFile:tCfg)
          endIf
        endIf

      break


      //回零
      case 274

        if TxtFile:bSync7Axis==false and TxtFile:bSync8Axis==false
          popUpMsg("同步七八轴未配置")
        else
          call UI:Control_YesNO("同步轴需要回零吗？",l_bRes)
          if l_bRes
            call UI:Control_PanelMd("同步轴正在回零")
            call ExtAxis:SingleMove(1,TxtFile:jHome,l_p,l_p,TxtFile:tCfg,mNomSpeed,l_trExtAxis)
            cls()
          endIf
        endIf
      break



      //上传
      case 276
        call UI:Control_YesNO("确定要上传吗?",l_bRes)
        if l_bRes
          call Kit:UpLoad()
          //return
        endIf
      break




      //保存
      case 277

        call UI:Control_YesNO("确定需要保存吗？",l_bRes)
        if l_bRes
          TxtFile:trSync7Axis.y=l_trExtAxis.x
          TxtFile:trSync8Axis.y=l_trExtAxis.y

          //   TxtFile:trSync7Axis.x=l_trExtAxis.rx
          //   TxtFile:trSync8Axis.x=l_trExtAxis.ry

          call TxtFile:SaveCfg(l_bRes)
          if l_bRes
            popUpMsg("保存成功")
          else
            popUpMsg("保存失败")
          endIf

        endIf
      break

      //
      case 278,255
        if l_trExtAxis.x!=TxtFile:trSync7Axis.y or  l_trExtAxis.y!=TxtFile:trSync8Axis.y
          call UI:Control_YesNO("参数未保存,确定需要退出吗？",l_bRes)
          if l_bRes
            cls()
            return
          endIf
        else
          cls()
          return
        endIf

      break


      case 270
        switch l_nIndex
          //          case 0
          ////            call UI:Sel_Edit(l_trExtAxis.rx,32,min(10,l_nIndex+1),l_sS)
          ////          break
          case 0
            call UI:Float_Edit(l_trExtAxis.x,32,min(10,l_nIndex+1))
          break

          //          case 2
          //            call UI:Sel_Edit(l_trExtAxis.ry,32,min(10,l_nIndex+1),l_sS)
          //          break

          case 1
            call UI:Float_Edit(l_trExtAxis.y,32,min(10,l_nIndex+1))
          break
        endSwitch

      break



    endSwitch



    //当前七轴位置
    if l_nKey!=-1 or !l_bFirst

      l_bFirst=true

      //××××××××××××××××××××××××××××


      //  sSItem[0]="七轴开启:"+l_sS[l_trExtAxis.rx]
      sSItem[0]="七轴home:"+toString(".3",l_trExtAxis.x)
      // sSItem[2]="八轴开启:"+l_sS[l_trExtAxis.ry]
      sSItem[1]="八轴home:"+toString("",l_trExtAxis.y)

      l_sBottom="参考,复位,记录,回零,,上传,保存,退出"


      call UI:Form_PanelList("LasMAN3.6->示教同步轴","同步轴",sSItem,l_nIndex,l_sBottom)




    endIf


    delay(0)

  endWhile

end

--- TeachTool.pgx ---
public program TeachTool()
  local bool l_bBool
begin
  //示教工具
  //1.两点法进行示教
  //2.使用不拆工具法示教
  if TxtFile:bTeachToolMode
    CalTool:bUpLoad=false
    call CalTool:start()
     if CalTool:bUpLoad
      TxtFile:tCfg=CalTool:tTool
      call TxtFile:SaveCfg(l_bBool)
       if !l_bBool
        popUpMsg("保存失败")
      endIf
      call Kit:UpLoad()
    endIf

  else
    call  Teach2Tool()

  endIf

end

--- TrajScreen.pgx ---
public program TrajScreen()
  local bool l_bRes
  local num l_nNum
begin

  //************************************************************
  cls()
  nApproIndex=0
  nCutIndex=0
  nLeaveIndex=0

  for l_nNum=0 to size(TxtFile:nPartTrajCount)-1
    TxtFile:nPartTrajCount[l_nNum]=0
  endFor


  //示教异步七轴
  if TxtFile:b7Axis
    //call Teach7Axis(TxtFile:trWorkplace.x,TxtFile:trWorkplace.y,1)
    if  (DataBase:nWorkPlaceIndex==1 and DataBase:bMutexAxis) or !DataBase:bMutexAxis
      //示教的时候把当前位置赋值给外部轴
      //2014.8.13
      if bFirstTeach==false
        call IO:GetAxis7Pos(TxtFile:trWorkplace.x,TxtFile:trAxisData.z)
        TxtFile:trWorkplace.y=nAxisSpeed
      endIf
      //×××××××××××××××
      call TeachAxis(TxtFile:trWorkplace.x,TxtFile:trWorkplace.y,TxtFile:trAxisData.z,TxtFile:trAxisData.rx,false)
    endIf
  endIf


  //示教异步八轴
  if TxtFile:b8Axis
    //  call Teach8Axis(TxtFile:trWorkplace.z,TxtFile:trWorkplace.rx,1)
    if (DataBase:bMutexAxis and DataBase:nWorkPlaceIndex==2) or !DataBase:bMutexAxis
      //示教的时候把当前位置赋值给外部轴
      //2014.8.13
      if bFirstTeach==false
        call IO:GetAxis8Pos(TxtFile:trWorkplace.z,TxtFile:trAxis8Data.z)
        TxtFile:trWorkplace.rx=nAxisSpeed
      endIf
      //××××××××××××××××××××××××
      call TeachAxis(TxtFile:trWorkplace.z,TxtFile:trWorkplace.rx,TxtFile:trAxis8Data.z,TxtFile:trAxis8Data.rx,true)
    endIf
  endIf



  //示教frame
  call UI:Control_YesNO("是否需要示教Frame",l_bRes)
  if l_bRes
    call TeachFrame(TxtFile:fTraj)
  endIf



  //示教的话则初始化点位
  if bFirstTeach==false
    resize(TxtFile:nTrajDelay,1,2)
    resize(TxtFile:pAppro,1,1)
    resize(TxtFile:bAppro,1,1)
    resize(TxtFile:jAppro,1,1)
    resize(TxtFile:trAppro,1,1)
    resize(TxtFile:trApproAxis,1,1)

    resize(TxtFile:pCut,1,sel(TxtFile:nSingleType==2 or TxtFile:nSingleType==23 or TxtFile:nSingleType==10  or TxtFile:nSingleType==20,1,3))
    resize(TxtFile:bMoveC,1,size(TxtFile:pCut,1))
    resize(TxtFile:pMoveC,1,size(TxtFile:pCut,1))
    resize(TxtFile:trCut,1,size(TxtFile:pCut,1))
    resize(TxtFile:trCutAxis,1,size(TxtFile:pCut,1))

    resize(TxtFile:pLeave,1,1)
    resize(TxtFile:bLeave,1,1)
    resize(TxtFile:jLeave,1,1)
    resize(TxtFile:trLeave,1,1)
    resize(TxtFile:trLeaveAxis,1,1)
    TxtFile:bLeave=TxtFile:bAppro=false

    TxtFile:trAppro={0,0,100,10,1,0}
    if TxtFile:nSingleType==10 or TxtFile:nSingleType==20
      TxtFile:trCut={1,0,100,5,1,0}
    else
      TxtFile:trCut={1,0,100,5,1,0}
    endIf
    TxtFile:trLeave={0,0,100,10,1,0}
    TxtFile:pAppro=TxtFile:pLeave=here(TxtFile:tCfg,TxtFile:fArray)
    TxtFile:jLeave=TxtFile:jAppro=herej()

    if TxtFile:nSingleType==2
      TxtFile:trDownLead={1,100,0,0,10,0}
    else
      TxtFile:trDownLead={1,100,0,0,0,0}
    endIf


    //××××××××××××××××××××××××××××××
    //2014.10.23
    //厚板切割
    //强制使用厚板切割程序
    if DataBase:bThickPlate
      TxtFile:trDownLead.y=101

    endIf
    //×××××××××××××××××××××××××××××××






    //激光延时默认
    //      TxtFile:trIODelay.x=0.3
    //      TxtFile:trIODelay.y=0

    TxtFile:nTrajDelay[0]=sel( TxtFile:bWeldEnable,0,0.3)
    TxtFile:nTrajDelay[1]=0
    for l_nNum=0 to size(TxtFile:pCut)-1

      TxtFile:pCut[l_nNum]=TxtFile:pMoveC[l_nNum]=here(TxtFile:tCfg,TxtFile:fArray)
      TxtFile:trCut[l_nNum]=TxtFile:trCut[0]
    endFor
    TxtFile:trWorkplace.rz=1
    //所有类型圆弧度
    TxtFile:trDownLead.rz=36
    //焊接
    TxtFile:trWorkplace.ry=5


    //为外部轴而设
    //205.03.23
    //外部轴程序修改
    if TxtFile:nSingleType==20 or TxtFile:nSingleType==9
      call ExtAxis:RecordExtAxis(TxtFile:trCutAxis[0],TxtFile:pCut[0].trsf,TxtFile:tCfg)
      TxtFile:pMoveC[0].trsf=TxtFile:pAppro[0].trsf=TxtFile:pLeave[0].trsf=TxtFile:pCut[0].trsf
      TxtFile:trApproAxis[0]=TxtFile:trLeaveAxis[0]=TxtFile:trCutAxis[0]
    endIf

    //2014.12.08
    //示教趋近与离开默认值

    TxtFile:trAppro=TxtFile:trLeave=DataBase:trTeachTemp

  endIf




  //把所有的点都给链接到相应的数值上
  for l_nNum=0 to size(TxtFile:pAppro)-1
    link(TxtFile:pAppro[l_nNum],TxtFile:fArray)
  endFor

  for l_nNum=0 to size(TxtFile:pLeave)-1
    link(TxtFile:pLeave[l_nNum],TxtFile:fArray)
  endFor

  for l_nNum=0 to size(TxtFile:pCut)-1
    link(TxtFile:pCut[l_nNum],TxtFile:fArray)
    link(TxtFile:pMoveC[l_nNum],TxtFile:fArray)
  endFor






  if TxtFile:nSingleType!=9

    nPointType=1
    while nPointType>=0 and nPointType<4

      switch nPointType
        //frame
        case 0
          call TeachFrame(TxtFile:fTraj)
        break

        //趋近点
        case 1
          call Approach()
        break

        //切割点
        case 2
          call Cut()
        break

        //离开点
        case 3
          call Leave()
        break

      endSwitch

    endWhile

  else

    call IdlePoint()

  endIf


  //******************************************************************************************



end

--- WeldTraj.pgx ---
program WeldTraj(bool& x_bRes)
  local num l_nId
  local num l_nBuffID
  local num l_nSize
  local num l_nNum
  local trsf l_trTrsf
begin
  //计算回退点
  l_nId=getMoveId()

  call Algorith:GetWeldReturn(TxtFile:pCut,TxtFile:pMoveC,TxtFile:bMoveC,l_nId,l_nBuffID,TxtFile:trIODelay.z,x_bRes)
  if !x_bRes or l_nBuffID<1  or l_nBuffID>(l_nId+0.0001)
   // popUpMsg(toString(".3",l_nBuffID))
    x_bRes=false
    return
  endIf

  if roundDown(l_nBuffID)==roundUp(l_nBuffID)
    l_nBuffID=l_nBuffID+0.0001
  endIf


  //圆弧

  if TxtFile:bMoveC[roundDown(l_nBuffID)]

    l_trTrsf=interpolateC(TxtFile:pCut[roundDown((l_nBuffID)-1)].trsf,TxtFile:pMoveC[roundDown(l_nBuffID)].trsf,TxtFile:pCut[roundDown(l_nBuffID)].trsf,l_nBuffID-roundDown(l_nBuffID))
  else

    l_trTrsf=interpolateL(TxtFile:pCut[roundDown((l_nBuffID)-1)].trsf,TxtFile:pCut[roundDown(l_nBuffID)].trsf,l_nBuffID-roundDown(l_nBuffID))
  endIf



  l_nSize=roundUp(l_nId)-roundDown(l_nBuffID)


  resize(TxtFile:jAppro,1,l_nSize)
  resize(TxtFile:pAppro,1,l_nSize)
  resize(TxtFile:trAppro,1,l_nSize)
  resize(TxtFile:bAppro,1,l_nSize)

  for l_nNum=0 to size(TxtFile:pAppro)-2
    TxtFile:bAppro[l_nNum]=true
    TxtFile:pAppro[l_nNum].trsf=TxtFile:pCut[roundDown(l_nId)-1-l_nNum].trsf
    TxtFile:trAppro[l_nNum]=TxtFile:trCut[roundDown(l_nId)-l_nNum-1]
  endFor

  TxtFile:pAppro[size(TxtFile:pAppro)-1].trsf=l_trTrsf
  TxtFile:bAppro[size(TxtFile:pAppro)-1]=true
  TxtFile:trAppro[size(TxtFile:pAppro)-1]=TxtFile:trAppro[0]

  for l_nNum=0 to roundDown(l_nBuffID)-2
    delete(TxtFile:pCut[0])
    delete(TxtFile:pMoveC[0])
    delete(TxtFile:trCut[0])
    delete(TxtFile:bMoveC[0])
  endFor
  TxtFile:pCut[0].trsf=l_trTrsf
  TxtFile:bMoveC[0]=false

  TxtFile:trPointCount.x=size(TxtFile:jAppro)
  TxtFile:trPointCount.y=size(TxtFile:pCut)

  x_bRes=true



end

--- WorkPlaceChose.pgx ---
public program WorkPlaceChose()
  local num l_nNum
begin
  //主要是在生产过程中对工位进行选择


  //生产程序一开启,变量初始化
  // DataBase:nWorkPlaceIndex=0
  //DataBase:nCycleIndex=0
  //DataBase:nWorkPlaceIndex ==1 表示工位1  ==2 表示工位2  ==3 表示工位3  ==4表示工位4
  //DataBase:nCycleIndex=1 表示生产第一个周期

  //参数强制合法化
  DataBase:nWorkPlaceCount=round(max(DataBase:nWorkPlaceCount,1))
  DataBase:nCycleCount=round(max(DataBase:nCycleCount,1))

  //进行判断是否生产结束
  if (DataBase:nWorkPlaceIndex>=DataBase:nWorkPlaceCount and DataBase:nCycleIndex==DataBase:nCycleCount) or DataBase:nCycleIndex>DataBase:nCycleCount
    DataBase:nInterfaceType=9
    DataBase:nWorkPlaceIndex=-1
    return
  endIf

  //按钮与常给信号的区别
  //




  //产品与工位选择
  //单个工位可以放多产品 一个工位最多可以放8个产品



  //单工位多产品
  if TxtFile:bMoreProd1Wp
    call GetProductMess("触发多工位")
    call OneWpMproChoose()
  else


    //六种触发方式
    call GetProductMess("等待按钮触发")
    switch DataBase:nCycleMode

      //按钮触发单工位：一个按钮一次
      case 0
        call IO:ProductReady(DataBase:nWorkPlaceIndex,false)
        call GetProductMess("工位按钮"+toString("",DataBase:nWorkPlaceIndex)+"触发")
      break


      //按钮触发单周期:一个按钮一个周期
      case 1

        DataBase:nWorkPlaceIndex=DataBase:nWorkPlaceIndex+1
        if DataBase:nWorkPlaceIndex>DataBase:nWorkPlaceCount
          DataBase:nWorkPlaceIndex=1
        endIf
        //等待IO
        if DataBase:nWorkPlaceIndex==1

          call IO:ProductReady(DataBase:nWorkPlaceIndex,true)
          DataBase:nCycleIndex=DataBase:nCycleIndex+1
          call GetProductMess("工位按钮"+toString("",DataBase:nWorkPlaceIndex)+"触发")
          call GetProductMess("开始执行周期"+toString("",DataBase:nCycleIndex))
        endIf


      break


      //按钮触发多周期:一个按钮多个周期
      case 2


        DataBase:nWorkPlaceIndex=DataBase:nWorkPlaceIndex+1
        if DataBase:nWorkPlaceIndex>DataBase:nWorkPlaceCount
          DataBase:nWorkPlaceIndex=1
          DataBase:nCycleIndex=DataBase:nCycleIndex+1
          call GetProductMess("开始执行周期"+toString("",DataBase:nCycleIndex))
        endIf
        //等待IO
        if DataBase:nWorkPlaceIndex==1 and DataBase:nCycleIndex==0
          call IO:ProductReady(DataBase:nWorkPlaceIndex,true)
          DataBase:nCycleIndex=DataBase:nCycleIndex+1
          call GetProductMess("工位按钮"+toString("",DataBase:nWorkPlaceIndex)+"触发")
          call GetProductMess("开始执行周期"+toString("",DataBase:nCycleIndex))
        endIf

      break

      //无按钮触发：没有按钮生产多周期
      case 3

        DataBase:nWorkPlaceIndex=DataBase:nWorkPlaceIndex+1
        if DataBase:nWorkPlaceIndex>DataBase:nWorkPlaceCount
          DataBase:nWorkPlaceIndex=1
          DataBase:nCycleIndex=DataBase:nCycleIndex+1
          call GetProductMess("开始执行周期"+toString("",DataBase:nCycleIndex))
        endIf
        if DataBase:nCycleIndex==0
          DataBase:nCycleIndex=1
          call GetProductMess("开始执行周期"+toString("",DataBase:nCycleIndex))
        endIf
      break

      //按钮触发排队
      //*********************************************
      //*********************************************
      case 4

        //最后一次按钮是OK
        while DataBase:nWorkPlaceButto==-1
          call IO:CanProduct(DataBase:nWorkPlaceButto)
          delay(0)
        endWhile
        DataBase:nWorkPlaceIndex=DataBase:nWorkPlaceButto
        DataBase:nWorkPlaceButto=-1
      break

      //**********************************************
      //
      //自定义触发方式
      //客户可以改写这里的代码
      case 5
        call Custom:ChooseCustomPro(DataBase:nWorkPlaceIndex,DataBase:nProductIndex)

      break

      //默认为报错
      default
        DataBase:nWorkPlaceIndex=-1
      break


    endSwitch
  endIf

  //工位等待时间
  if DataBase:nWorkPlaceIndex>0 and DataBase:nWorkPlaceIndex<=DataBase:nWorkPlaceCount

    if TxtFile:trIODelay.rx>0
      call GetProductMess("工位等待"+toString(".1",TxtFile:trIODelay.rx)+"秒")
      delay(max(TxtFile:trIODelay.rx,0))
    endIf
  endIf

end
